{attribute clr [Container(Layout.Tabs)]}
TYPE
    ProcessData EXTENDS TcoEntityBase :
    STRUCT

        {attribute addProperty Name "<#Entity header#>"}
        EntityHeader : EntityHeader     := (Parent := THISSTRUCT);
		{attribute addProperty Name "<#CU00x#>"}
		{attribute clr [Container(Layout.Stack)]}
        CU00x : CU00xProcessData := (Parent := THISSTRUCT);
		
//		
    END_STRUCT
END_TYPE

(* stored: Version 1.1.0.1
   DUT ProcessData: Id {113396d1-0fe0-4862-b140-87fe92cd116d} *)
